// TIA Portal V20 export
VAR_GLOBAL   // PLC tag table "Default tag table"
   "BA010AZCRBK05.02" AT %I1016.2 : Bool;   // COMPENSATOR LIMIT SENSOR(-)
   "BA010AZCRBK05.03" AT %I1016.3 : Bool;   // COMPENSATOR LIMIT SENSOR(+)
   "BA010AZCRBK05.12" AT %I1017.2 : Bool;   // COMPENSATOR HOMING SENSOR
   "BA010AZCRBK06.03" AT %I1020.3 : Bool;   // NG & MANUAL INPUT LIMIT SENSOR(-)
   "BA010AZCRBK06.04" AT %I1020.4 : Bool;   // NG & MANUAL INPUT LIMIT SENSOR(+)
   "BA010AZCRBK06.05" AT %I1020.5 : Bool;   // NG & MANUAL INPUT MAGAZINE LIMIT SENSOR(-)
   "BA010AZCRBK06.06" AT %I1020.6 : Bool;   // NG & MANUAL INPUT MAGAZINE LIMIT SENSOR(+)
   "BA010AZCRBK06.13" AT %I1021.3 : Bool;   // NG & MANUAL INPUT HOMING SENSOR
   "BA010AZCRBK06.15" AT %I1021.5 : Bool;   // NG & MANUAL INPUT MAGAZINE HOMING SENSOR
   "BA010AZCRBK07.00" AT %I1024.0 : Bool;   // POSITION MOVING LIMIT SENSOR(-)
   "BA010AZCRBK07.01" AT %I1024.1 : Bool;   // POSITION MOVING LIMIT SENSOR(+)
   "BA010AZCRBK07.02" AT %I1024.2 : Bool;   // VISION HOMING SENSOR
   "BA010AZCRBK07.03" AT %I1024.3 : Bool;   // ELECTRODE NG KICKER HOMING SENSOR
   "BA010AZCRBK07.10" AT %I1025.0 : Bool;   // POSITION MOVING HOMING SENSOR
   "BA010AZCRBK07.11" AT %I1025.1 : Bool;   // CUTTER HOMING SENSOR
   "BA010AZCRBK07.13" AT %I1025.3 : Bool;   // ELECTRODE PASS KICKER HOMING SENSOR
   "BA010AZCRSP506.00" AT %I3300.0 : Bool;   // TAB DETECTION SENSOR
   "BA010AZCRSP506.01" AT %I3300.1 : Bool;   // TAPE DETECTION SENSOR
   "BA010AZCRSP506.04" AT %Q3300.0 : Bool;   // OutputCam_FeedingRollAxisB
   "BA010AZCRSP506.05" AT %Q3300.1 : Bool;   // OutputCam_ElectrodeCutterAxisZ
   "BA010AZCRSP506.07" AT %Q3300.3 : Bool;   // OutputCam_NgKickerAxisZ
   "BA010AZCRSP506.08" AT %Q3300.4 : Bool;   // SPARE
   "BA010AZCRSP507.04" AT %Q3350.0 : Bool;   // OutputCam_PassKickerAxisZ
   "BA010AZCRSP507.05" AT %Q3350.1 : Bool;   // SPARE
   "BA010AZCRSP507.06" AT %Q3350.2 : Bool;   // SPARE
   "BA010AZCRSP507.07" AT %Q3350.3 : Bool;   // SPARE
   "BA010AZCRSP507.08" AT %Q3350.4 : Bool;   // SPARE
   BA010AZCRDR4_FeedingRollAxisB_Actor_Interface_TorqueDataAddressIn AT %I5434.0 : "PD_TEL750_IN";
   BA010AZCRDR5_ElectordCutterAxisZ_Actor_Interface_TorqueDataAddressIn AT %I5534.0 : "PD_TEL750_IN";
   BA010AZCRDR6_PositionMovingAxisX_Actor_Interface_TorqueDataAddressIn AT %I5644.0 : "PD_TEL750_IN";
   BA020AZCRDR7_NgManualInputAxisY_Actor_Interface_TorqueDataAddressIn AT %I5734.0 : "PD_TEL750_IN";
   BA020AZCRDR8_MagazineAxisZ_Actor_Interface_TorqueDataAddressIn AT %I5844.0 : "PD_TEL750_IN";
   BA020AZCRDR9_VisionAxisZ_Actor_Interface_TorqueDataAddressIn AT %I5944.0 : "PD_TEL750_IN";
   BA020AZCRDR10_NgKickerAxisZ_Actor_Interface_TorqueDataAddressIn AT %I6044.0 : "PD_TEL750_IN";
   BA020AZCRDR11_PassKickerAxisZ_Actor_Interface_TorqueDataAddressIn AT %I6144.0 : "PD_TEL750_IN";
   BA010AZCRDR4_FeedingRollAxisB_Actor_Interface_TorqueDataAddressOut AT %Q5434.0 : "PD_TEL750_OUT";
   BA010AZCRDR5_ElectordCutterAxisZ_Actor_Interface_TorqueDataAddressOut AT %Q5534.0 : "PD_TEL750_OUT";
   BA010AZCRDR6_PositionMovingAxisX_Actor_Interface_TorqueDataAddressOut AT %Q5644.0 : "PD_TEL750_OUT";
   BA020AZCRDR7_NgManualInputAxisY_Actor_Interface_TorqueDataAddressOut AT %Q5734.0 : "PD_TEL750_OUT";
   BA020AZCRDR8_MagazineAxisZ_Actor_Interface_TorqueDataAddressOut AT %Q5844.0 : "PD_TEL750_OUT";
   BA020AZCRDR9_VisionAxisZ_Actor_Interface_TorqueDataAddressOut AT %Q5944.0 : "PD_TEL750_OUT";
   BA020AZCRDR10_NgKickerAxisZ_Actor_Interface_TorqueDataAddressOut AT %Q6044.0 : "PD_TEL750_OUT";
   BA020AZCRDR11_PassKickerAxisZ_Actor_Interface_TorqueDataAddressOut AT %Q6144.0 : "PD_TEL750_OUT";
END_VAR
